{region '#Template'}
	{attribute 'Category' := 'H'}
	{attribute 'Version' := '0.0.1.0'}
	{attribute 'Tags' := 'H, Plant, HtgCir, Heating circuit'}
	{attribute 'Description' := 'Heizkreis	// Heating circuit'}
{endregion}
FUNCTION_BLOCK FB_BA_H_HtgCir01 EXTENDS FB_BA_View
VAR_INPUT
END_VAR
VAR_OUTPUT
	eOpMod 					: E_BA_EnergyLvl;
	bRls					: BOOL;	
	fSp    					: REAL;
	bPu    					: BOOL;
	fVlv   					: REAL;
END_VAR
VAR_INPUT CONSTANT
	TFl						: FB_BA_SensorAnalog_IO;												
	TRt						: FB_BA_SensorAnalog_IO;																									
	Vlv						: FB_BA_Vlv;									
	Pu						: FB_BA_Pu1st;	
	Sp						: FB_BA_H_HtgCir_Sp;												
	OpMod					: FB_BA_H_OpMod;									
	HtgLmt					: FB_BA_HtgLmt;							
	TFlCtrl					: FB_BA_PID;
	GeneralSettings			: FB_BA_RawSubscriber;		
	stGeneralSettings		: ST_BA_GeneralSettings;	
END_VAR
VAR
	PlantLock				: FB_BA_PlantLock := (iParent := THIS^);
	
END_VAR
VAR // added by the converter: edge detectors and wires of the graphical bodies
    _w1 : ANY;
END_VAR

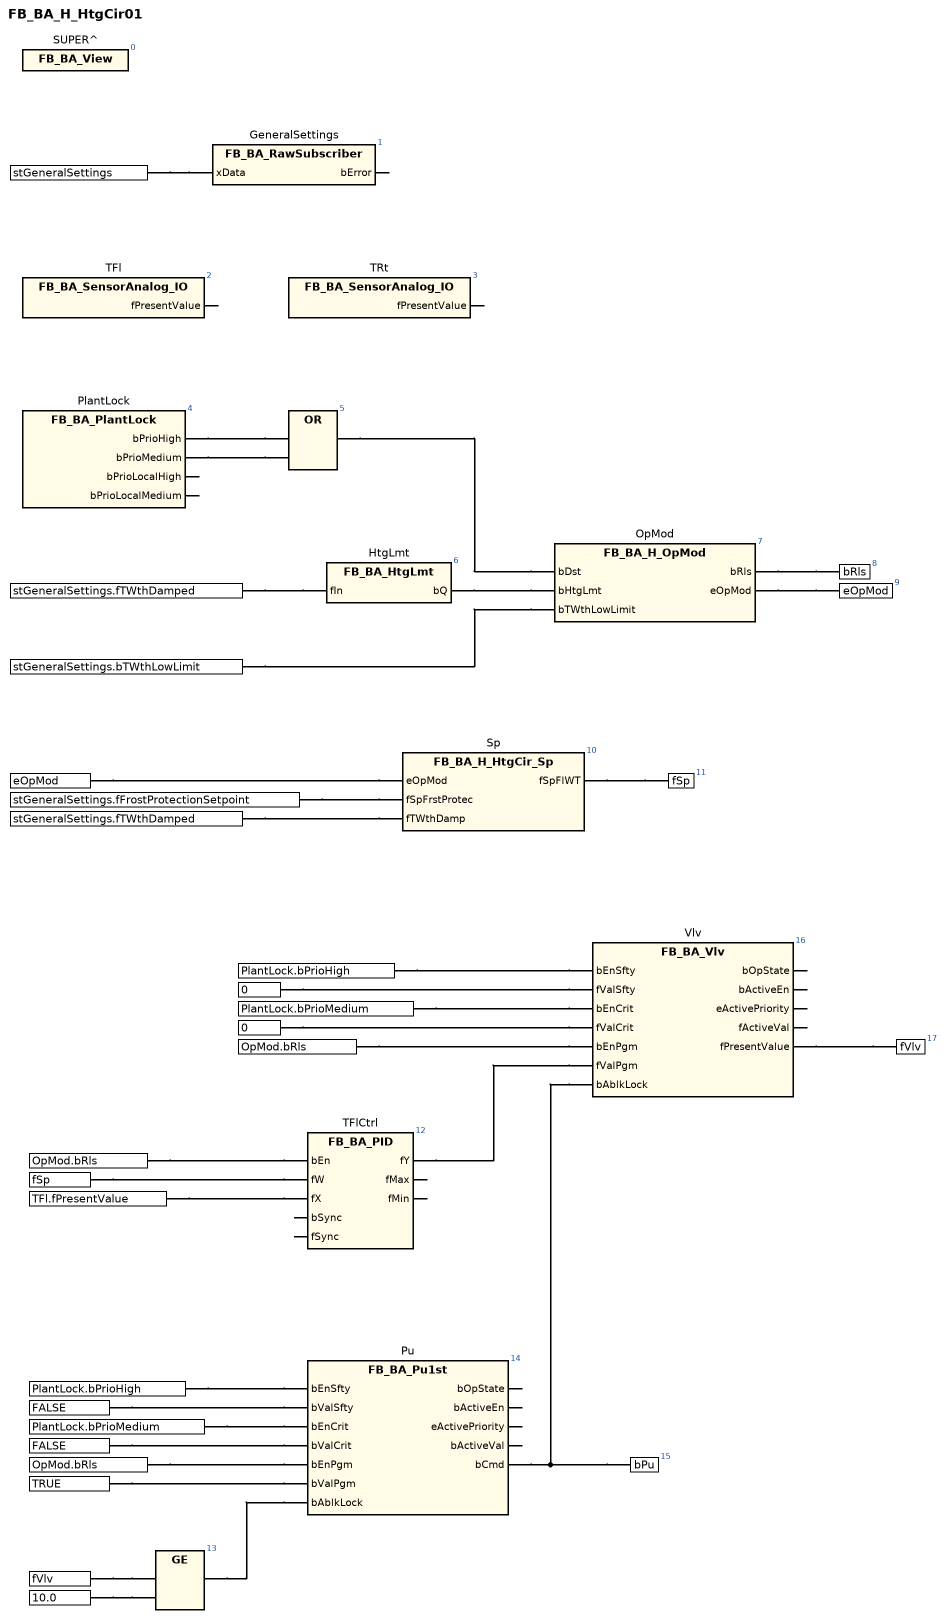
// note: 14 stored wires end on pins the file does not list and are not shown
SUPER^(); // FB_BA_View
GeneralSettings(xData := stGeneralSettings); // FB_BA_RawSubscriber
TFl(); // FB_BA_SensorAnalog_IO
TRt(); // FB_BA_SensorAnalog_IO
PlantLock(); // FB_BA_PlantLock
_w1 := PlantLock.bPrioHigh OR PlantLock.bPrioMedium;
HtgLmt(fIn := stGeneralSettings.fTWthDamped); // FB_BA_HtgLmt
OpMod(bDst := _w1, bHtgLmt := HtgLmt.bQ, bTWthLowLimit := stGeneralSettings.bTWthLowLimit); // FB_BA_H_OpMod
bRls := OpMod.bRls;
eOpMod := OpMod.eOpMod;
Sp(
    eOpMod := eOpMod,
    fSpFrstProtec := stGeneralSettings.fFrostProtectionSetpoint,
    fTWthDamp := stGeneralSettings.fTWthDamped); // FB_BA_H_HtgCir_Sp
fSp := Sp.fSpFlWT;
TFlCtrl(bEn := OpMod.bRls, fW := fSp, fX := TFl.fPresentValue); // FB_BA_PID
Pu(
    bEnSfty := PlantLock.bPrioHigh,
    bValSfty := FALSE,
    bEnCrit := PlantLock.bPrioMedium,
    bValCrit := FALSE,
    bEnPgm := OpMod.bRls,
    bValPgm := TRUE,
    bAblkLock := fVlv >= 10.0); // FB_BA_Pu1st
bPu := Pu.bCmd;
Vlv(
    bEnSfty := PlantLock.bPrioHigh,
    fValSfty := 0,
    bEnCrit := PlantLock.bPrioMedium,
    fValCrit := 0,
    bEnPgm := OpMod.bRls,
    fValPgm := TFlCtrl.fY,
    bAblkLock := Pu.bCmd); // FB_BA_Vlv
fVlv := Vlv.fPresentValue;

METHOD FB_init : BOOL
VAR_INPUT
	bInitRetains : BOOL; // if TRUE, the retain variables are initialized (warm start / cold start)
	bInCopyCode : BOOL;  // if TRUE, the instance afterwards gets moved into the copy code (online change)
END_VAR
TFl.iParent								:= THIS^;		
TFl.iLabel 								:= LblCmpHeating.H_HtgCir_TFl;	
TFl.sObjectName							:= '{Idx=01}';	
TFl.eDPADMode							:= E_BA_DPADMode.eInclude;																																	
TFl.MV.eUnit							:= E_BA_Unit.eTemperature_DegreesCelsius;
TFl.MV.eEnPlantLock						:= E_BA_LockPriority.eMedium;
TFl.MV.fResolution 						:= 0.01;
TFl.MV.fScaleOffset 					:= 0; 

TRt.iParent								:= THIS^;		
TRt.iLabel 								:= LblCmpHeating.H_HtgCir_TRt;	
TRt.sObjectName							:= '{Idx=01}';														
TRt.eDPADMode							:= E_BA_DPADMode.eInclude;																																	
TRt.MV.eUnit							:= E_BA_Unit.eTemperature_DegreesCelsius;
TRt.MV.eEnPlantLock						:= E_BA_LockPriority.eNoLock;
TRt.MV.fResolution 						:= 0.01;
TRt.MV.fScaleOffset 					:= 0;  
				
Vlv.iParent								:= THIS^;	
Vlv.iLabel								:= LblCmpHeating.H_HtgCir_Vlv;
Vlv.sObjectName							:= '{Idx=01}';										 
Vlv.eDPADMode							:= E_BA_DPADMode.eInclude;									
				
Pu.iParent								:= THIS^;
Pu.iLabel								:= LblCmpHeating.H_HtgCir_Pu;
Pu.sObjectName							:= '{Idx=01}';										 
Pu.eDPADMode							:= E_BA_DPADMode.eInclude;				
				
Sp.iParent								:= THIS^;	
Sp.iLabel								:= LblCmpHeating.H_HtgCir_Sp;
Sp.sObjectName							:= '{Idx=01}';										 
Sp.eDPADMode							:= E_BA_DPADMode.eInclude;												
				
OpMod.iParent							:= THIS^;	
OpMod.iLabel							:= LblCmpHeating.H_HtgCir_OpMod;
OpMod.sObjectName						:= '{Idx=01}';										 
OpMod.eDPADMode							:= E_BA_DPADMode.eInclude;									
				
HtgLmt.iParent							:= THIS^;	
HtgLmt.iLabel							:= LblCmpHeating.H_HtgCir_HtgLmt;
HtgLmt.sObjectName						:= '{Idx=01}';										 
HtgLmt.eDPADMode						:= E_BA_DPADMode.eInclude;

TFlCtrl.iParent							:= THIS^;
TFlCtrl.iLabel							:= LblCmpHeating.H_HtgCir_TFlCtrl;
TFlCtrl.sObjectName						:= '{Idx=01}';
TFlCtrl.eDPADMode						:= E_BA_DPADMode.eInclude;																																	
TFlCtrl.Ctrl.eOutputUnit				:= E_BA_Unit.eOther_Percent;
TFlCtrl.Ctrl.eActionRm					:= E_BA_Action.eReverse;
TFlCtrl.Ctrl.fMinOutputRm				:= 0;
TFlCtrl.Ctrl.fMaxOutputRm				:= 100;
TFlCtrl.Ctrl.fProportionalConstant		:= 3;
TFlCtrl.Ctrl.fIntegralConstant			:= 180;

GeneralSettings.Subject					:= Site.GeneralSettings_Subject;
GeneralSettings.sTarget					:= Site.GeneralSettings_NetId;
END_METHOD

END_FUNCTION_BLOCK

(* stored: Version 1.1.0.1, ProductVersion 3.1.4024.6
   POU FB_BA_H_HtgCir01: Id {eb068529-9d74-4ea0-b70a-b3ed0424e738}, SpecialFunc None
   Method FB_init: Id {316fd3be-1bf1-4183-b0e0-0cd1012c472a} *)
